Staubli VAL3: getTrajItem.pgx

public program getTrajItem(TrajectoryItem& x_tTrajItem[], num x_nIndex)
begin
  //
  // get all the FIELD
  //
  x_tTrajItem=jEditPoint.tData[x_nIndex].tSuper
end
